(* PLC project robin.project, CODESYS CODESYS V3.5 SP15 *)
(* stored: creationDateTime 2019-11-25T16:48:00.9238887, modificationDateTime 2019-11-25T16:42:20.5256552 *)

TYPE TestStruct_foo : STRUCT
  var_bool_1 : BOOL := TRUE;
  var_struct_1 : TestSubStruct;  (* var_bool_2 : BOOL := TRUE; *)
  var_struct_2 : TestSubStruct;
END_STRUCT;
END_TYPE

TYPE TestSubStruct : STRUCT
  var_float64_1 : LREAL := 0.123456789;
  var_float64_2 : LREAL := -10.9876554321;
END_STRUCT;
END_TYPE

TYPE TestStruct_bar : STRUCT
  var_bool : BOOL := TRUE;
  var_byte : BYTE := 128;
  var_int16 : INT := -12345;
  var_uint64 : ULINT := 9876543210123456789;
  var_float32 : REAL := 1234.5;
  var_float64 : LREAL := 0.123456789;
  var_struct : TestSubStruct;
END_STRUCT;
END_TYPE

TYPE TestStruct_arr : STRUCT
  var_string : STRING(30);
  var_float64_array : ARRAY[1..10] OF LREAL;  (* var_int16_array : ARRAY[1..Robin.DEF_ARRAY_LEN] OF INT; // not usefull *)
  var_bytemultiarray : ByteMultiArray;
END_STRUCT;
END_TYPE

FUNCTION_BLOCK Robin
  VAR CONSTANT
    MAX_SIZE : INT := 10;
    SEM_TIMEOUT : UDINT := 1000;  (* in ms (16#FFFFFFFF = inf) *)
  END_VAR
  VAR_OUTPUT CONSTANT
    DEF_ARRAY_LEN : INT := 20;
  END_VAR
  VAR
    data : ARRAY[1..MAX_SIZE] OF RobinData;
    idx : UINT;
    i : INT;
  END_VAR

            idx := 1;

          

(* FB_Init is always available implicitly and it is used primarily for initialization. The return value is not evaluated. For a specific influence, you can also declare the methods explicitly and provide additional code there with the standard initialization code. You can evaluate the return value. *)
METHOD FB_Init : BOOL
  VAR_INPUT
    bInitRetains : BOOL;  (* TRUE: the retain variables are initialized (reset warm / reset cold) *)
    bInCopyCode : BOOL;  (* TRUE: the instance will be copied to the copy code afterward (online change) *)
  END_VAR
                  FOR i := 1 TO MAX_SIZE DO
	data[i].sem := RTS_INVALID_HANDLE;
	data[i].shm := RTS_INVALID_HANDLE;
END_FOR;

                
END_METHOD

(* FB_Exit must be implemented explicitly. If there is an implementation, then the method is called before the controller removes the code of the function block instance (implicit call). The return value is not evaluated. *)
METHOD FB_Exit : BOOL
  VAR_INPUT
    bInCopyCode : BOOL;  (* TRUE: the exit method is called in order to leave the instance which will be copied afterwards (online change). *)
  END_VAR
                  // IF NOT bInCopyCode THEN
// 	result := SysSemProcessEnter(sem, SEM_TIMEOUT);
	FOR i := 1 TO MAX_SIZE DO
		IF data[idx].shm <> RTS_INVALID_HANDLE THEN
			data[idx].result := SysSharedMemoryClose(data[idx].shm);
// 			data[idx].result := SysSharedMemoryDelete(data[idx].shm);
		END_IF
	END_FOR;
// 	result := SysSharedMemoryDelete(shm);
// 	result := SysSemProcessDelete(sem);
// END_IF

                
END_METHOD

METHOD open : BOOL
  VAR_INPUT
    name : STRING;
    size : __UXINT;
  END_VAR
                  IF data[idx].shm = RTS_INVALID_HANDLE THEN
	data[idx].shm := SysSharedMemoryOpen2(name, 0, ADR(size), ADR(data[idx].result));
	IF data[idx].shm <> RTS_INVALID_HANDLE THEN
		data[idx].sem := SysSemProcessCreate(name, ADR(data[idx].result));
		IF data[idx].sem <> RTS_INVALID_HANDLE THEN
			open := TRUE;
		END_IF
	ELSE
		open := FALSE;
	END_IF
ELSE
	open := TRUE;
END_IF

                
END_METHOD

{attribute 'hasanytype'}
METHOD read
  VAR_INPUT
    name : STRING;
    {attribute 'anytypeclass' := 'ANY'}
    var_ : __SYSTEM.AnyType;
  END_VAR
  VAR
    size : __UXINT := DINT_TO___UXINT(var_.diSize);
  END_VAR
                  IF open(name, size) THEN
	IF SysSemProcessEnter(data[idx].sem, SEM_TIMEOUT) = Errors.ERR_OK THEN
		data[idx].bytes := SysSharedMemoryRead(data[idx].Shm, 0, var_.pValue, size, ADR(data[idx].result));
		data[idx].result := SysSemProcessLeave(data[idx].sem);
	END_IF
END_IF
idx := idx + 1;

                
END_METHOD

{attribute 'hasanytype'}
METHOD write
  VAR_INPUT
    name : STRING;
    {attribute 'anytypeclass' := 'ANY'}
    var_ : __SYSTEM.AnyType;
  END_VAR
  VAR
    size : __UXINT := DINT_TO___UXINT(var_.diSize);
  END_VAR
                  IF open(name, size) THEN
	IF SysSemProcessEnter(data[idx].sem, SEM_TIMEOUT) = Errors.ERR_OK THEN
		data[idx].bytes := SysSharedMemoryWrite(data[idx].shm, 0, var_.pValue, size, ADR(data[idx].result));
		data[idx].result := SysSemProcessLeave(data[idx].sem);
	END_IF
END_IF
idx := idx + 1;

                
END_METHOD
END_FUNCTION_BLOCK

PROGRAM ROS_PRG
  VAR_INPUT
    double_to_ros : LREAL;
    struct_to_ros : TestStruct_foo;
    string_to_ros : STRING;
    double_flarray_to_ros : ARRAY[1..5] OF LREAL;
    {attribute 'robin_var_len'}
    double_vlarray_to_ros : ARRAY[1..5] OF LREAL;
  END_VAR
  VAR_OUTPUT
    double_to_codesys : LREAL;
    struct_to_codesys : TestStruct_foo;
    string_to_codesys : STRING;
    double_flarray_to_codesys : ARRAY[1..5] OF LREAL;
    {attribute 'robin_var_len'}
    double_vlarray_to_codesys : ARRAY[1..5] OF LREAL;
  END_VAR
  VAR
    robin : Robin;
  END_VAR

                    robin();
robin.read('double_to_codesys', double_to_codesys);
robin.read('struct_to_codesys', struct_to_codesys);
robin.read('string_to_codesys', string_to_codesys);
robin.read('double_flarray_to_codesys', double_flarray_to_codesys);
robin.read('double_vlarray_to_codesys', double_vlarray_to_codesys);
// robin.read('struct_to_codesys_arr', struct_to_codesys_arr);
robin.write('double_to_ros', double_to_ros);
robin.write('struct_to_ros', struct_to_ros);
robin.write('string_to_ros', string_to_ros);
robin.write('double_flarray_to_ros', double_flarray_to_ros);
robin.write('double_vlarray_to_ros', double_vlarray_to_ros);
// robin.write('struct_to_ros_arr', struct_to_ros_arr);

                  
END_PROGRAM

PROGRAM MAIN

                    ROS_PRG.double_to_ros := ROS_PRG.double_to_codesys;
ROS_PRG.struct_to_ros := ROS_PRG.struct_to_codesys;
ROS_PRG.string_to_ros := ROS_PRG.string_to_codesys;
ROS_PRG.double_flarray_to_ros := ROS_PRG.double_flarray_to_codesys;
ROS_PRG.double_vlarray_to_ros := ROS_PRG.double_vlarray_to_codesys;
// ROS_PRG.struct_to_ros_arr := ROS_PRG.struct_to_codesys_arr;

                  
END_PROGRAM

CONFIGURATION Device
  RESOURCE Application ON PLC
    {attribute 'qualified_only'}
    VAR_GLOBAL  (* GVL *)
      double_to_ros : LREAL;
    END_VAR
    TASK MainTask(INTERVAL := T#10ms, PRIORITY := 1);
    PROGRAM MAIN WITH MainTask : MAIN;
    PROGRAM ROS_PRG WITH MainTask : ROS_PRG;
  END_RESOURCE
END_CONFIGURATION

CONFIGURATION SoftMotion General Axis Pool
END_CONFIGURATION
